ABB RobotStudio station: First Behaviour.rspag

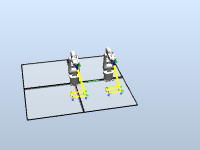
--- station ---
Station Multirobots - ABB (saved by RobotStudio 6.8.8307.1040)
Controller Robot2, task T_ROB1: task frame (RAPID world) sits at (0, 700, 0) mm in the station
Controller Robot1
  mechanical unit ROB_1: IRB120_3_58__01, 6 joints, base frame (0, 0, 0) mm
Controller Robot2
  mechanical unit ROB_1: IRB120_3_58__01_2, 6 joints, base frame (0, 0, 0) mm
Layout (positions relative to the parent item):
  - IRB120_3_58__01 [mechanism, from Robots\IRB120_3_58_G_01.rslib] at (0, 0, 0) mm; joint values [0, 0, 0, 0, 0.5236, 0] (rad or m)
  - IRB120_3_58__01_2 [mechanism, from Robots\IRB120_3_58_G_01.rslib] at (0, 700, 0) mm; joint values [0, 0, 0, 0, 0.5236, 0] (rad or m)
Station logic (signal -> signal, property => property):
  Robot1.arrival1 -> Robot2.arrival1
  Robot2.arrival2 -> Robot1.arrival2

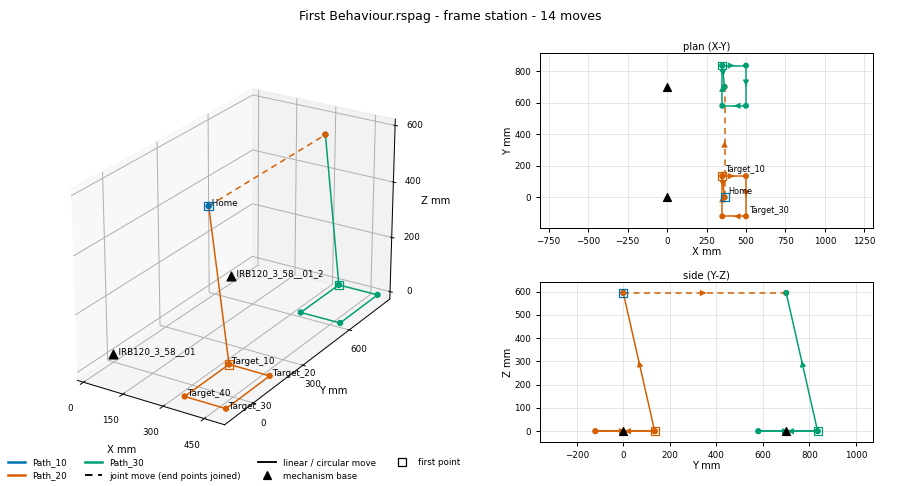
[picture p0: tool path of First Behaviour.rspag in frame station, 14 of 14 moves have a stored position in this frame; points joined in program order, loops and branches not executed]
--- Backups/Robot1/RAPID/TASK1/PROGMOD/Module1.mod ---
MODULE Module1
	CONST robtarget Home:=[[364.353829072,0,594],[0.5,0,0.866025404,0],[0,0,0,0],[9E+09,9E+09,9E+09,9E+09,9E+09,9E+09]];
    CONST robtarget Target_10:=[[350,135,0],[0,0,1,0],[0,0,0,0],[9E+09,9E+09,9E+09,9E+09,9E+09,9E+09]];
    CONST robtarget Target_20:=[[500,135,0],[0,0,1,0],[0,0,0,0],[9E+09,9E+09,9E+09,9E+09,9E+09,9E+09]];
    CONST robtarget Target_30:=[[500,-120,0],[0,0,1,0],[0,0,0,0],[9E+09,9E+09,9E+09,9E+09,9E+09,9E+09]];
    CONST robtarget Target_40:=[[350,-120,0],[0,0,1,0],[0,0,0,0],[9E+09,9E+09,9E+09,9E+09,9E+09,9E+09]];

    PROC main()
        SetDo arrival1, 0;          !reestablecer valor de variable

        Path_10;                    !Trayectoria a Home
        SetDO arrival1, 1;          !Indicacion de fin de tarea con variable

        WaitDI arrival2, 1;         !Espera hasta que el otro robot indique que ha acabado
        Path_20;                    !Trayectoria del rectangulo

    ENDPROC

	PROC Path_10()
	    MoveJ Home,v200,fine,tool0\WObj:=wobj0;
	ENDPROC
    PROC Path_20()
        MoveL Target_10,v200,z0,tool0\WObj:=wobj0;
        MoveL Target_20,v200,z0,tool0\WObj:=wobj0;
        MoveL Target_30,v200,z0,tool0\WObj:=wobj0;
        MoveL Target_40,v200,z0,tool0\WObj:=wobj0;
        MoveL Target_10,v200,z0,tool0\WObj:=wobj0;
        MoveL Home,v200,z100,tool0\WObj:=wobj0;
    ENDPROC
ENDMODULE

--- Backups/Robot2/RAPID/TASK1/PROGMOD/Module1.mod ---
MODULE Module1
	CONST robtarget Home:=[[364.353826402,0,593.999995375],[0.499999968,0,0.866025422,0],[-1,0,-1,0],[9E+09,9E+09,9E+09,9E+09,9E+09,9E+09]];
    CONST robtarget Target_10:=[[350,135,0],[0,0,1,0],[0,0,0,0],[9E+09,9E+09,9E+09,9E+09,9E+09,9E+09]];
    CONST robtarget Target_20:=[[500,135,0],[0,0,1,0],[0,0,0,0],[9E+09,9E+09,9E+09,9E+09,9E+09,9E+09]];
    CONST robtarget Target_30:=[[500,-120,0],[0,0,1,0],[0,0,0,0],[9E+09,9E+09,9E+09,9E+09,9E+09,9E+09]];
    CONST robtarget Target_40:=[[350,-120,0],[0,0,1,0],[0,0,0,0],[9E+09,9E+09,9E+09,9E+09,9E+09,9E+09]];


    PROC main()
        SetDo arrival2, 0;          !reestablecer valor de variable

        Path_20;                    !Trayectoria a Home
        SetDo arrival2, 1;          !Indicacion de fin de tarea con variable

        WaitDI arrival1, 1;         !Espera hasta que el otro robot indique que ha acabado
        Path_30;                    !Trayectoria del rectangulo

    ENDPROC

    PROC Path_20()
	    MoveJ Home,v200,fine,tool0\WObj:=wobj0;
	ENDPROC
    PROC Path_30()
        MoveL Target_10,v200,z0,tool0\WObj:=wobj0;
        MoveL Target_20,v200,z0,tool0\WObj:=wobj0;
        MoveL Target_30,v200,z0,tool0\WObj:=wobj0;
        MoveL Target_40,v200,z0,tool0\WObj:=wobj0;
        MoveL Target_10,v200,z0,tool0\WObj:=wobj0;
        MoveL Home,v200,z100,tool0\WObj:=wobj0;
    ENDPROC
ENDMODULE

--- Backups/Robot1/SYSPAR/EIO.cfg ---
EIO:CFG_1.0:6:1::
#
EIO_SIGNAL:

      -Name "arrival1" -SignalType "DO" -Access "All"

      -Name "arrival2" -SignalType "DI"

--- Backups/Robot2/SYSPAR/EIO.cfg ---
EIO:CFG_1.0:6:1::
#
EIO_SIGNAL:

      -Name "arrival1" -SignalType "DI"

      -Name "arrival2" -SignalType "DO" -Access "All"
